SYSTEM System (* System Configuration *)
  (* Standard: 61499-1 *)
  (* Version 0.0, 1/9/2024, Cheyan, Schneider Electric *)
  {SET_ATTRIBUTE(System.Device.FolderPath, EcoRT_0)}
  APPLICATION APP1
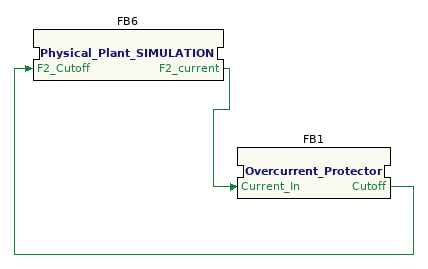
    (* Plant (Power System) *)
    (* Control (IEC 61499) *)
    (* Feeder 2 *)
    FBS
      FB6 : Physical_Plant_SIMULATION;
      FB1 : Overcurrent_Protector;
    END_FBS
    ADAPTER_CONNECTIONS
      FB1.Cutoff TO FB6.F2_Cutoff;
      FB6.F2_current TO FB1.Current_In;
    END_CONNECTIONS
  END_APPLICATION
  DEVICE EcoRT_0 : Soft_dPAC
    RESOURCE RES0 : EMB_RES_ECO
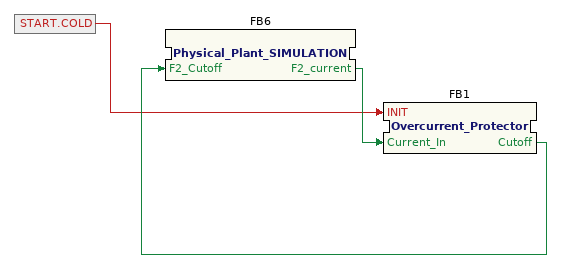
      FBS
        FB6 : Physical_Plant_SIMULATION;
        FB1 : Overcurrent_Protector;
      END_FBS
      EVENT_CONNECTIONS
        START.COLD TO FB1.INIT;
      END_CONNECTIONS
      ADAPTER_CONNECTIONS
        FB1.Cutoff TO FB6.F2_Cutoff;
        FB6.F2_current TO FB1.Current_In;
      END_CONNECTIONS
    END_RESOURCE
  END_DEVICE
  MAPPINGS
    APP1.FB6 ON EcoRT_0.RES0;
    APP1.FB1 ON EcoRT_0.RES0;
  END_MAPPINGS
END_SYSTEM
